// TIA Portal V20 export
DATA_BLOCK "Instance_FB_Get_In_Rework_Conveyor_Belt_DB"   // DB110
// stored: AutoNumber false, InstanceOfName FB_Get_In_Rework_Conveyor_Belt, InstanceOfType FB
"FB_Get_In_Rework_Conveyor_Belt"
   // VAR_INPUT
   //    Emergency_Stop_Release : Bool;
   //    Start : Bool;
   //    Sensor_Water_Fountain_Exit_Functional_Test_Spinner_Conveyor_Belt : Bool;
   //    Sensor_Spinner_Exit_Functional_Test_Position_Withdrawn : Bool;
   //    Sensor_Spinner_Exit_Functional_Test_Position_Advanced : Bool;
   //    Sensor_Water_Fountain_Geting_Entrace_Rework_Conveyor_Belt_Start : Bool;
   //    Sensor_Water_Fountain_Geting_Entrace_Rework_Conveyor_Belt_Finish : Bool;
   // END_VAR
   // VAR_OUTPUT
   //    Turn_On_Conveyor_Belt_Motor_Rework_Conveyor_Belt_Get_Exit_Funcional_Test : Bool;
   // END_VAR
BEGIN
END_DATA_BLOCK
